//==================================================================================================
//								RJM Maszyny sp. z o.o.
//									04.06.2022
//	Obsługa czujnika  NO
// 	v1.0	|| TC v 3.1.4024.22		|| - pierwsza wersja
//==================================================================================================
FUNCTION_BLOCK FB_Czujnik_NO IMPLEMENTS ITF_Czujnik
VAR_INPUT
	bSymulacja								: BOOL;
END_VAR
VAR
	bWejscie						AT %I*	: BOOL;
END_VAR

//==================================================================================================
//								RJM Maszyny sp. z o.o.
//									13.05.2022
//	Informacja czy czujnik jest zadziałany 
// 	v1.0	|| TC v 3.1.4024.22		|| - pierwsza wersja
//==================================================================================================
PROPERTY CzyZadzialany : BOOL
GET
CzyZadzialany								:= bWejscie;
END_GET
END_PROPERTY

END_FUNCTION_BLOCK

(* stored: Version 1.1.0.1, ProductVersion 3.1.4024.11
   POU FB_Czujnik_NO: Id {a309e5c5-49d5-4f4a-94f9-421545786459}, SpecialFunc None
   Property CzyZadzialany: Id {acf3546f-68a9-47d1-b1c1-b4e2e1b0ec7a}
   Get Get: Id {b5827c71-7ea6-4b81-bf27-2ae7e097e936} *)
